// TwinCAT 3 PLC project AnalysisPLC
// ProgramVersion: 3.1.4023.0
// libraries:
//   Tc2_EtherCAT, * (Beckhoff Automation GmbH)
//   Tc2_Standard, * (Beckhoff Automation GmbH)
//   Tc2_System, * (Beckhoff Automation GmbH)
//   Tc2_Utilities, * (Beckhoff Automation GmbH)
//   Tc3_Analytics, * (Beckhoff Automation GmbH)
//   Tc3_EventLogger, * (Beckhoff Automation GmbH)
//   Tc3_Module, * (Beckhoff Automation GmbH)
// project tree:
//   / AnalyticsTask.TcTTO, AnalyticsTask_V1_C1.TcTTO, PlcTask.TcTTO
//   DUTs/Analytics/ E_AnalysisComponents.TcDUT, E_DataSourceState.TcDUT, ST_AnalysisReset.TcDUT
//   DUTs/Analytics/HMI/DataSourcePage/ ST_HMI_DataSourceConfig.TcDUT, ST_HMI_DataSourceCtrl.TcDUT, ST_HMI_DataSourceHist.TcDUT, ST_HMI_DataSourceHistInfo.TcDUT, ST_HMI_DataSourceHistRecordInfo.TcDUT, ST_HMI_DataSourceLive.TcDUT, ST_HMI_DataSourceStream.TcDUT
//   DUTs/Analytics/HMI/ ST_HMI_MapItem.TcDUT, ST_HMI_N1_Network.TcDUT, ST_KeyValuePair.TcDUT
//   GVLs/ Analytics.TcGVL, AnalyticsHMI.TcGVL
//   POUs/Analytics/DataSource/Interfaces/ I_DataSource.TcIO, I_VirtualInputSource.TcIO
//   POUs/Analytics/DataSource/Interfaces/VirtualInputSources/ I_V1_Virtual_Input_Source_1.TcIO
//   POUs/Analytics/DataSource/T01 DataSource/ FB_T1_DataSource.TcPOU
//   POUs/Analytics/ FB_Analysis.TcPOU
//   POUs/Analytics/Networks/N01 Network/ FB_N1_Network.TcPOU
//   POUs/Analytics/Networks/N01 Network/Modules/ FB_N1_M1_LifetimeAnalysis1Ch.TcPOU, FB_N1_M2_ThresholdStringClassifier1Ch.TcPOU, FB_N1_M3_TrendLine.TcPOU
//   POUs/Analytics/[Helper]/ F_AlyTimestampToDCTimestruct.TcPOU, F_AlyTimestampToFileTime.TcPOU, F_DCTimestructToFileTime.TcPOU, F_FileTimeToDCTimestruct.TcPOU
//   POUs/ MAIN.TcPOU, MAIN_Analytics.TcPOU, MAIN_Analytics_V1_C1.TcPOU

CONFIGURATION AnalysisPLC
    RESOURCE PLC ON TwinCAT3
        TASK AnalyticsTask(INTERVAL := T#10ms, PRIORITY := 21);
        TASK AnalyticsTask_V1_C1(INTERVAL := T#10ms, PRIORITY := 1);
        TASK PlcTask(INTERVAL := T#10ms, PRIORITY := 20);
        PROGRAM MAIN_Analytics WITH AnalyticsTask : MAIN_Analytics;
        PROGRAM MAIN_Analytics_V1_C1 WITH AnalyticsTask_V1_C1 : MAIN_Analytics_V1_C1;
        PROGRAM MAIN WITH PlcTask : MAIN;
    END_RESOURCE
END_CONFIGURATION

// ---- DUTs/Analytics/E_AnalysisComponents.TcDUT
{attribute 'qualified_only'}
{attribute 'strict'}
TYPE E_AnalysisComponents : 
(
	All := -1,
	N1_Network := 0,
	N1_M1_LifetimeAnalysis1Ch := 1,
	N1_M2_ThresholdStringClassifier1Ch := 2,
	N1_M3_TrendLine := 3
) ;
END_TYPE

// ---- DUTs/Analytics/E_DataSourceState.TcDUT
{attribute 'qualified_only'}
{attribute 'strict'}
TYPE E_DataSourceState : 
(
	eUnknown := 0,
	eNotConnected,
	eReceiveData,
	eReceiveData_Cancel,
	eReceiveData_Pause,
	eError
) ;
END_TYPE

// ---- DUTs/Analytics/HMI/DataSourcePage/ST_HMI_DataSourceConfig.TcDUT
TYPE ST_HMI_DataSourceConfig : 
STRUCT
	nID: DINT;
	sName: STRING(80);
	sDisplayName: STRING(80);
	nStreamCount: INT;
	aStreams: ARRAY [0..9] OF ST_HMI_DataSourceStream;
END_STRUCT
END_TYPE

// ---- DUTs/Analytics/HMI/DataSourcePage/ST_HMI_DataSourceCtrl.TcDUT
TYPE ST_HMI_DataSourceCtrl : 
STRUCT
	nActiveMachineIdx: INT;
	nActiveStreamIdx: INT;
	
	bHistorical: BOOL;
	
	//IF Historical
	nActiveRecordIdx: INT;
	
	dtSelectedRangeStart: DCTIMESTRUCT;
	dtSelectedRangeEnd: DCTIMESTRUCT;
	
	bStart: BOOL;
	bCancel: BOOL;
	bPause: BOOL;
	
	bUpdateRecordList: BOOL;
END_STRUCT
END_TYPE

// ---- DUTs/Analytics/HMI/DataSourcePage/ST_HMI_DataSourceHist.TcDUT
TYPE ST_HMI_DataSourceHist : 
STRUCT
	dtCurrentTimestamp: DCTIMESTRUCT;
	nCurrentRecordID: DINT;
	sDisplayName: STRING(80);
	stSourceInfo: ST_HMI_DataSourceHistInfo;
	nRecordCount: DINT;
	aRecords: ARRAY [0..255] OF ST_HMI_DataSourceHistRecordInfo;
END_STRUCT
END_TYPE

// ---- DUTs/Analytics/HMI/DataSourcePage/ST_HMI_DataSourceHistInfo.TcDUT
TYPE ST_HMI_DataSourceHistInfo : 
STRUCT
	sSPGuid: GUID;
	sAlyFilePath: STRING(255);
	sSourceType: STRING(80);
	sTopic: STRING(255);
	sLayoutID: GUID;
END_STRUCT
END_TYPE

// ---- DUTs/Analytics/HMI/DataSourcePage/ST_HMI_DataSourceHistRecordInfo.TcDUT
TYPE ST_HMI_DataSourceHistRecordInfo : 
STRUCT
	nID: DINT;
	sName: STRING(80);
	sDisplayName: STRING(80);
	dtRecordStart: DCTIMESTRUCT;
	dtRecordEnd: DCTIMESTRUCT;
	dtSelectedRangeStart: DCTIMESTRUCT;
	dtSelectedRangeEnd: DCTIMESTRUCT;
END_STRUCT
END_TYPE

// ---- DUTs/Analytics/HMI/DataSourcePage/ST_HMI_DataSourceLive.TcDUT
TYPE ST_HMI_DataSourceLive : 
STRUCT
	dtLiveTimestamp: DCTIMESTRUCT;
	sDisplayName: STRING(80);
END_STRUCT
END_TYPE

// ---- DUTs/Analytics/HMI/DataSourcePage/ST_HMI_DataSourceStream.TcDUT
TYPE ST_HMI_DataSourceStream : 
STRUCT
	sSource: STRING(80);
	sStreamSystemID: GUID;
	sTopic: STRING(255);
	stLive: ST_HMI_DataSourceLive;
	stHist: ST_HMI_DataSourceHist;
END_STRUCT
END_TYPE

// ---- DUTs/Analytics/HMI/ST_HMI_MapItem.TcDUT
TYPE ST_HMI_MapItem : 
STRUCT
	sName: T_MaxString;
	sDescription: T_MaxString;
	sPosition: T_MaxString;
	nStatus: INT;
END_STRUCT
END_TYPE

// ---- DUTs/Analytics/HMI/ST_HMI_N1_Network.TcDUT
TYPE ST_HMI_N1_Network : 
STRUCT
	//Lifetime Analysis 1Ch
	tM1_fbLifetimeElapsed: ST_ALY_TimeSpan; //Elapsed (Times)
	tM1_fbLifetimeRemaining: ST_ALY_TimeSpan; //Remaining (Times)
	
	//Threshold String Classifier 1Ch
	sM2_sStringLevel1: STRING(255); //ConfigLevel1
	sM2_sStringLevel2: STRING(255); //ConfigLevel2
	sM2_sStringLevel3: STRING(255); //ConfigLevel3
	sM2_sResult: STRING(255); //String Classification
	fM2_nDataIn: LREAL; //Value
	
	//Trend Line
	aM3_aTrendData: ARRAY [1..1] OF ARRAY [1..10080] OF LREAL; //RawData
	dtM3_fbLastValue: DCTIMESTRUCT; //LastValueTimestamp
	nM3_nCountValues: DINT; //CountedValues
	aM3_aChannelNames: ARRAY [0..0] OF STRING(255); //DisplayNames
END_STRUCT
END_TYPE

// ---- DUTs/Analytics/HMI/ST_KeyValuePair.TcDUT
TYPE ST_KeyValuePair : 
STRUCT
	sKey: STRING(255);
	sValue: STRING(255);
END_STRUCT
END_TYPE

// ---- DUTs/Analytics/ST_AnalysisReset.TcDUT
TYPE ST_AnalysisReset : 
STRUCT
	eResetComponent: E_AnalysisComponents := E_AnalysisComponents.All;
	bResetExecute: BOOL;
END_STRUCT
END_TYPE

// ---- GVLs/Analytics.TcGVL
{attribute 'qualified_only'}
VAR_GLOBAL
	//DataSources
	fbT1_DataSource: FB_T1_DataSource;
	
	bLock_T1: BOOL;
	
	stReset: ST_AnalysisReset;
END_VAR

// ---- GVLs/AnalyticsHMI.TcGVL
{attribute 'qualified_only'}
VAR_GLOBAL
	//Switch between historical and live data
	stHMI_DataSourceCtrl: ST_HMI_DataSourceCtrl;
	stHMI_DataSourceConfig: ARRAY [0..0] OF ST_HMI_DataSourceConfig := [
											(nID:= 1, sName:= 'fbT1_DataSource', sDisplayName:= 'b375d0e8-9412-9d91-04c5-b1a76c1b6bbd', nStreamCount:= 1,
												aStreams:=[(sSource:= 'TwinCAT Analytics Logger', sStreamSystemID:= STRING_TO_GUID('b375d0e8-9412-9d91-04c5-b1a76c1b6bbd'), sTopic:= 'DefaultMainTopic/PlcStream1',
													stLive:= (sDisplayName:= 'DataSource T1')
														)])
											];
	
	//Reset
	
	//HMI Structs
	stHMI_N1_Network: ST_HMI_N1_Network;
	
	//HMI Map Items
	aMapItems: ARRAY [0..0] OF ST_HMI_MapItem := [(sName:='b375d0e8-9412-9d91-04c5-b1a76c1b6bbd', sDescription:='', sPosition:='', nStatus:= 0)];
END_VAR

// ---- POUs/Analytics/DataSource/Interfaces/I_DataSource.TcIO
INTERFACE I_DataSource

METHOD Call : BOOL
END_METHOD

METHOD GetData : BOOL
VAR_INPUT
	nElement: UDINT;
END_VAR
END_METHOD

METHOD HistoricalCtrl : BOOL
VAR_INPUT
	stCtrl: REFERENCE TO ST_HMI_DataSourceCtrl;
	stHistStreamInfo: REFERENCE TO ST_HMI_DataSourceHist;
	stRecordInfo: REFERENCE TO ST_HMI_DataSourceHistRecordInfo;
END_VAR
END_METHOD

METHOD UpdateRecordList : BOOL
VAR_INPUT
	stCtrl: REFERENCE TO ST_HMI_DataSourceCtrl;
	sStreamSystemID: GUID;
	stHistStreamInfo: REFERENCE TO ST_HMI_DataSourceHist;
END_VAR
END_METHOD

METHOD NewDataAvailable : BOOL
VAR_INPUT
	nLastDataHandle: ULINT;
END_VAR
END_METHOD

PROPERTY nDataHandle : ULINT
GET
END_GET
END_PROPERTY

PROPERTY nElements : UDINT
GET
END_GET
END_PROPERTY

PROPERTY dtTimestamp : DCTIMESTRUCT
GET
END_GET
END_PROPERTY

END_INTERFACE

// ---- POUs/Analytics/DataSource/Interfaces/I_VirtualInputSource.TcIO
INTERFACE I_VirtualInputSource

PROPERTY tTimestamp : ULINT
GET
END_GET
END_PROPERTY

PROPERTY bNewData : BOOL
GET
END_GET
END_PROPERTY

END_INTERFACE

// ---- POUs/Analytics/DataSource/Interfaces/VirtualInputSources/I_V1_Virtual_Input_Source_1.TcIO
INTERFACE I_V1_Virtual_Input_Source_1 EXTENDS I_VirtualInputSource

PROPERTY bV1_Virtual_Input : BOOL
GET
END_GET
END_PROPERTY

PROPERTY nV1_Virtual_Input_1 : INT
GET
END_GET
END_PROPERTY

END_INTERFACE

// ---- POUs/MAIN_Analytics.TcPOU
PROGRAM MAIN_Analytics
VAR
	sCurrentStreamSystemID: GUID;
	stHistStreamInfo: REFERENCE TO ST_HMI_DataSourceHist;
	stHistRecordInfo: REFERENCE TO ST_HMI_DataSourceHistRecordInfo;
END_VAR



//Call DataSource FBs
IF MAIN_Analytics_V1_C1.nLastDataHandle = Analytics.fbT1_DataSource.nDataHandle THEN
	Analytics.fbT1_DataSource.Call();
END_IF



//Map to HMI
CASE AnalyticsHMI.stHMI_DataSourceCtrl.nActiveMachineIdx OF
	0:
		MAIN_Analytics_V1_C1.A_MapToHMI();
END_CASE

END_PROGRAM

// ---- POUs/MAIN_Analytics_V1_C1.TcPOU
PROGRAM MAIN_Analytics_V1_C1
VAR_OUTPUT
	bError: BOOL;
	ipTcResult: I_TcMessage;
	nLastDataHandle: ULINT;
END_VAR
VAR
	fbAnalysis: FB_Analysis;
	
	nElement: UDINT;
	nSample: UDINT;
END_VAR

IF TestAndSet(Analytics.bLock_T1) THEN
	IF Analytics.fbT1_DataSource.NewDataAvailable(nLastDataHandle) THEN
		FOR nElement:= 1 TO Analytics.fbT1_DataSource.nElements BY 1 DO
			IF Analytics.fbT1_DataSource.GetData(nElement) THEN

				fbAnalysis.Call(Analytics.fbT1_DataSource);
				IF fbAnalysis.bError THEN
					EXIT;
				END_IF
			END_IF
		END_FOR
		nLastDataHandle:= Analytics.fbT1_DataSource.nDataHandle;
	ELSE
		fbAnalysis.Call(0);
	END_IF
	Analytics.bLock_T1:= FALSE;
END_IF

//Error Handling
bError:= fbAnalysis.bError;
ipTcResult:= fbAnalysis.ipTcResult;

ACTION A_MapToHMI:

//Map HMI Current Timestamp
AnalyticsHMI.stHMI_DataSourceConfig[0].aStreams[0].stLive.dtLiveTimestamp:= Analytics.fbT1_DataSource.dtTimestamp;

//Map In-/Outputs of the Analysis to HMI Structs
fbAnalysis.fbN1_Network.SetHMIValues(ADR(AnalyticsHMI.stHMI_N1_Network));
END_ACTION

END_PROGRAM

// ---- POUs/Analytics/FB_Analysis.TcPOU
FUNCTION_BLOCK FB_Analysis
VAR_INPUT
	fbN1_Network: FB_N1_Network;
END_VAR
VAR_OUTPUT
	bError: BOOL;
	ipTcResult: I_TcMessage;
END_VAR
VAR
	R_TRIG_Reset: R_TRIG;
	bResetBusy: BOOL;
	
	_tTimestamp: ULINT;
END_VAR

METHOD Call : BOOL
VAR_INPUT
	ipVirtual_Input_Source_1: I_V1_Virtual_Input_Source_1;
END_VAR
VAR
END_VAR

IF ipVirtual_Input_Source_1 <> 0 THEN

	_tTimestamp:= ipVirtual_Input_Source_1.tTimestamp;

	//Analytics Network "Network" with ID: 1
	fbN1_Network.Call(ipVirtual_Input_Source_1);


	//Error Handling
	IF fbN1_Network.bError THEN
		bError:= TRUE;
		ipTcResult:= fbN1_Network.ipTcResult;
	ELSE
		bError:= FALSE;
	END_IF
END_IF
END_METHOD

PROPERTY tTimestamp : ULINT
GET
tTimestamp:= _tTimestamp;
END_GET
END_PROPERTY

END_FUNCTION_BLOCK

// ---- POUs/Analytics/Networks/N01 Network/FB_N1_Network.TcPOU
//Analytics Network "Network" with ID: 1
{attribute 'no_assign'}
FUNCTION_BLOCK FB_N1_Network
VAR_INPUT
	fbM1_LifetimeAnalysis1Ch: FB_N1_M1_LifetimeAnalysis1Ch;
	fbM2_ThresholdStringClassifier1Ch: FB_N1_M2_ThresholdStringClassifier1Ch;
	fbM3_TrendLine: FB_N1_M3_TrendLine;
END_VAR
VAR_OUTPUT
	bError: BOOL;
	ipTcResult: I_TcMessage;
END_VAR
VAR
END_VAR

METHOD Call : BOOL
VAR_INPUT
	ipVirtual_Input_Source_1: I_V1_Virtual_Input_Source_1;
END_VAR
VAR
END_VAR

ValueMapping(ipVirtual_Input_Source_1);

//The Lifetime Analysis 1Ch calculates the elapsed and the estimated remaining lifetime of a device. The input channel should provide boolean values so that every switching procedure represents a cycle which can be converted into the elapsed lifetime. Optional a boolean signal for Enable Execution can be selected, so that the algorithm is just active if the value of the selected signal is TRUE.
fbM1_LifetimeAnalysis1Ch.Call(SEL(ipVirtual_Input_Source_1 <> 0, FALSE, ipVirtual_Input_Source_1.bNewData));

//The Threshold String Classifier 1Ch classifies the input values into three different classes according to the configured thresholds. The class names (output strings) can be configured individually as String 1, String 2 and String 3. Optional a boolean signal for Enable Execution can be selected, so that the algorithm is just active if the value of the selected signal is TRUE.
fbM2_ThresholdStringClassifier1Ch.Call(SEL(ipVirtual_Input_Source_1 <> 0, FALSE, ipVirtual_Input_Source_1.bNewData));

//This Module is used for the One-click Dashboard to generate a special analytics trend chart.
fbM3_TrendLine.Call(SEL(ipVirtual_Input_Source_1 <> 0, FALSE, ipVirtual_Input_Source_1.bNewData));

//Error Handling
IF fbM1_LifetimeAnalysis1Ch.bError THEN
	bError:= TRUE;
	ipTcResult:= fbM1_LifetimeAnalysis1Ch.ipTcResult;
ELSIF fbM2_ThresholdStringClassifier1Ch.bError THEN
	bError:= TRUE;
	ipTcResult:= fbM2_ThresholdStringClassifier1Ch.ipTcResult;
ELSIF fbM3_TrendLine.bError THEN
	bError:= TRUE;
	ipTcResult:= fbM3_TrendLine.ipTcResult;
ELSE
	bError:= FALSE;
END_IF
END_METHOD

METHOD Reset : BOOL
VAR
	bResult: BOOL := TRUE;
END_VAR

bResult:= bResult AND fbM1_LifetimeAnalysis1Ch.Reset();
bResult:= bResult AND fbM2_ThresholdStringClassifier1Ch.Reset();
bResult:= bResult AND fbM3_TrendLine.Reset();
Reset:= bResult;
END_METHOD

METHOD SetHMIValues : BOOL
VAR_INPUT
	pHMI_N1_Network: POINTER TO ST_HMI_N1_Network;
END_VAR
VAR
END_VAR

//Modules
fbM1_LifetimeAnalysis1Ch.SetHMI(pHMI_N1_Network);
fbM2_ThresholdStringClassifier1Ch.SetHMI(pHMI_N1_Network);
fbM3_TrendLine.SetHMI(pHMI_N1_Network);

SetHMIValues:= TRUE;
END_METHOD

METHOD PRIVATE ValueMapping : BOOL
VAR_INPUT
	ipVirtual_Input_Source_1: I_V1_Virtual_Input_Source_1;
END_VAR
VAR
END_VAR
//Module fbM1_LifetimeAnalysis1Ch
fbM1_LifetimeAnalysis1Ch.tTimestamp:= ipVirtual_Input_Source_1.tTimestamp;
fbM1_LifetimeAnalysis1Ch.bDataIn:= ipVirtual_Input_Source_1.bV1_Virtual_Input;

//Module fbM2_ThresholdStringClassifier1Ch
fbM2_ThresholdStringClassifier1Ch.tTimestamp:= ipVirtual_Input_Source_1.tTimestamp;
fbM2_ThresholdStringClassifier1Ch.nDataIn:= ipVirtual_Input_Source_1.nV1_Virtual_Input_1;

//Module fbM3_TrendLine
fbM3_TrendLine.tTimestamp:= ipVirtual_Input_Source_1.tTimestamp;
fbM3_TrendLine.nDataInCh1:= ipVirtual_Input_Source_1.nV1_Virtual_Input_1;
END_METHOD

END_FUNCTION_BLOCK

// ---- POUs/Analytics/Networks/N01 Network/Modules/FB_N1_M1_LifetimeAnalysis1Ch.TcPOU
//The Lifetime Analysis 1Ch calculates the elapsed and the estimated remaining lifetime of a device. The input channel should provide boolean values so that every switching procedure represents a cycle which can be converted into the elapsed lifetime. Optional a boolean signal for Enable Execution can be selected, so that the algorithm is just active if the value of the selected signal is TRUE.
FUNCTION_BLOCK FB_N1_M1_LifetimeAnalysis1Ch
VAR_INPUT
	bDataIn: BOOL;
	tTimestamp: ULINT;
	bEnableExecution: BOOL := TRUE;
	bReset: BOOL;
	bReconfigure: BOOL := TRUE;
	stThresholdLevel: ST_ALY_Threshold;
	tLifetimeEstimated: LTIME;
END_VAR
VAR_OUTPUT
	bError: BOOL;
	ipTcResult: I_TcMessage;
	bNewResult: BOOL;
	fbLifetimeElapsed: FB_ALY_TimeSpan;
	fbLifetimeRemaining: FB_ALY_TimeSpan;
END_VAR
VAR
	
	bConfigured: BOOL;
	R_TRIG_Reconfigure: R_TRIG;
	
	fbALY_LifeTimeAnalysis_1Ch: FB_ALY_LifeTimeAnalysis_1Ch;
END_VAR

METHOD Call : BOOL
VAR_INPUT
	bNewData: BOOL;
END_VAR
VAR
END_VAR
IF NOT bConfigured THEN
	bConfigured:= TRUE;

	tLifetimeEstimated:= LTIME#1h;

	//stThresholdLevel
	stThresholdLevel.eComparisonOperator:= E_ALY_ComparisonOperator.NotEqualTo;
	stThresholdLevel.fThreshold:= 0;

END_IF

R_TRIG_Reconfigure(CLK:= bReconfigure);
IF R_TRIG_Reconfigure.Q THEN
	fbALY_LifeTimeAnalysis_1Ch.ConfigureChannel(stThresholdLevel:=stThresholdLevel);

	fbALY_LifeTimeAnalysis_1Ch.Configure(tLifetimeEstimated:=tLifetimeEstimated);

	bReconfigure:= FALSE;
END_IF

IF bReset THEN
	Reset();
END_IF

IF bEnableExecution THEN
	IF bNewData THEN
		fbALY_LifeTimeAnalysis_1Ch.SetChannelValue(Input:=bDataIn);

		fbALY_LifeTimeAnalysis_1Ch.Call(tTimestamp:=tTimestamp);

		bNewResult:= fbALY_LifeTimeAnalysis_1Ch.bNewResult;
		fbLifetimeElapsed:= fbALY_LifeTimeAnalysis_1Ch.fbLifetimeElapsed;
		fbLifetimeRemaining:= fbALY_LifeTimeAnalysis_1Ch.fbLifetimeRemaining;

		bError:= fbALY_LifeTimeAnalysis_1Ch.bError;
		ipTcResult:= fbALY_LifeTimeAnalysis_1Ch.ipResultMessage;
	END_IF
END_IF
END_METHOD

METHOD Reset : BOOL
VAR
END_VAR
Reset:= fbALY_LifeTimeAnalysis_1Ch.Reset();

bNewResult:= fbALY_LifeTimeAnalysis_1Ch.bNewResult;
fbLifetimeElapsed:= fbALY_LifeTimeAnalysis_1Ch.fbLifetimeElapsed;
fbLifetimeRemaining:= fbALY_LifeTimeAnalysis_1Ch.fbLifetimeRemaining;

bError:= NOT Reset;
ipTcResult:= fbALY_LifeTimeAnalysis_1Ch.ipResultMessage;
END_METHOD

METHOD SetHMI : BOOL
VAR_INPUT
	pHMI_N1_Network: POINTER TO ST_HMI_N1_Network;
END_VAR
VAR
END_VAR

pHMI_N1_Network^.tM1_fbLifetimeElapsed:= fbLifetimeElapsed.stStructured;
pHMI_N1_Network^.tM1_fbLifetimeRemaining:= fbLifetimeRemaining.stStructured;
END_METHOD

END_FUNCTION_BLOCK

// ---- POUs/Analytics/Networks/N01 Network/Modules/FB_N1_M2_ThresholdStringClassifier1Ch.TcPOU
//The Threshold String Classifier 1Ch classifies the input values into three different classes according to the configured thresholds. The class names (output strings) can be configured individually as String 1, String 2 and String 3. Optional a boolean signal for Enable Execution can be selected, so that the algorithm is just active if the value of the selected signal is TRUE.
FUNCTION_BLOCK FB_N1_M2_ThresholdStringClassifier1Ch
VAR_INPUT
	nDataIn: INT;
	tTimestamp: ULINT;
	bEnableExecution: BOOL := TRUE;
	bReset: BOOL;
	bReconfigure: BOOL := TRUE;
	fThresholdLevel12: LREAL;
	fThresholdLevel23: LREAL;
	sStringLevel1: STRING(255);
	sStringLevel2: STRING(255);
	sStringLevel3: STRING(255);
END_VAR
VAR_OUTPUT
	bError: BOOL;
	ipTcResult: I_TcMessage;
	bNewResult: BOOL;
	sResult: STRING(255);
	fbTimeLastEvent: FB_ALY_DateTime;
END_VAR
VAR
	
	bConfigured: BOOL;
	R_TRIG_Reconfigure: R_TRIG;
	
	fbALY_ThresholdStringClassificator_1Ch: FB_ALY_ThresholdStringClassificator_1Ch;
END_VAR

METHOD Call : BOOL
VAR_INPUT
	bNewData: BOOL;
END_VAR
VAR
END_VAR
IF NOT bConfigured THEN
	bConfigured:= TRUE;

	fThresholdLevel12:= 20000;
	fThresholdLevel23:= 28000;
	sStringLevel1:= 'Normal';
	sStringLevel2:= 'High';
	sStringLevel3:= 'High High';

END_IF

R_TRIG_Reconfigure(CLK:= bReconfigure);
IF R_TRIG_Reconfigure.Q THEN
	fbALY_ThresholdStringClassificator_1Ch.Configure(
		fThresholdLevel12:= fThresholdLevel12,
		fThresholdLevel23:= fThresholdLevel23,
		sStringLevel1:= sStringLevel1,
		sStringLevel2:= sStringLevel2,
		sStringLevel3:= sStringLevel3);

	bReconfigure:= FALSE;
END_IF

IF bReset THEN
	Reset();
END_IF

IF bEnableExecution THEN
	IF bNewData THEN
		fbALY_ThresholdStringClassificator_1Ch.SetChannelValue(Input:=nDataIn);

		fbALY_ThresholdStringClassificator_1Ch.Call(tTimestamp:=tTimestamp);

		bNewResult:= fbALY_ThresholdStringClassificator_1Ch.bNewResult;
		sResult:= fbALY_ThresholdStringClassificator_1Ch.sResult;
		fbTimeLastEvent:= fbALY_ThresholdStringClassificator_1Ch.fbTimeLastEvent;

		bError:= fbALY_ThresholdStringClassificator_1Ch.bError;
		ipTcResult:= fbALY_ThresholdStringClassificator_1Ch.ipResultMessage;
	END_IF
END_IF
END_METHOD

METHOD Reset : BOOL
VAR
END_VAR
Reset:= fbALY_ThresholdStringClassificator_1Ch.Reset();

bNewResult:= fbALY_ThresholdStringClassificator_1Ch.bNewResult;
sResult:= fbALY_ThresholdStringClassificator_1Ch.sResult;
fbTimeLastEvent:= fbALY_ThresholdStringClassificator_1Ch.fbTimeLastEvent;

bError:= NOT Reset;
ipTcResult:= fbALY_ThresholdStringClassificator_1Ch.ipResultMessage;
END_METHOD

METHOD SetHMI : BOOL
VAR_INPUT
	pHMI_N1_Network: POINTER TO ST_HMI_N1_Network;
END_VAR
VAR
END_VAR

pHMI_N1_Network^.sM2_sStringLevel1:= sStringLevel1;
pHMI_N1_Network^.sM2_sStringLevel2:= sStringLevel2;
pHMI_N1_Network^.sM2_sStringLevel3:= sStringLevel3;
pHMI_N1_Network^.sM2_sResult:= sResult;
pHMI_N1_Network^.fM2_nDataIn:= TO_LREAL(nDataIn);
END_METHOD

END_FUNCTION_BLOCK

// ---- POUs/Analytics/Networks/N01 Network/Modules/FB_N1_M3_TrendLine.TcPOU
//This Module is used for the One-click Dashboard to generate a special analytics trend chart.
FUNCTION_BLOCK FB_N1_M3_TrendLine
VAR_INPUT
	nDataInCh1: INT;
	tTimestamp: ULINT;
	bEnableExecution: BOOL := TRUE;
	bReset: BOOL;
	bReconfigure: BOOL := TRUE;
	aChannelNames: ARRAY [0..0] OF STRING(255);
END_VAR
VAR_OUTPUT
	bError: BOOL;
	ipTcResult: I_TcMessage;
	bNewResult: BOOL;
	aTrendData: ARRAY [1..1] OF ARRAY [1..10080] OF LREAL;
	fbLastValue: FB_ALY_DateTime;
	nCountValues: UDINT;
END_VAR
VAR
	nNumChannels: INT := 1;
	
	bConfigured: BOOL;
	R_TRIG_Reconfigure: R_TRIG;
	
	fbALY_TrendLine: FB_ALY_TrendLine(nNumChannels:=nNumChannels);
END_VAR

METHOD Call : BOOL
VAR_INPUT
	bNewData: BOOL;
END_VAR
VAR
END_VAR
IF NOT bConfigured THEN
	bConfigured:= TRUE;

	aChannelNames[0]:= 'Resistor';

END_IF

R_TRIG_Reconfigure(CLK:= bReconfigure);
IF R_TRIG_Reconfigure.Q THEN

	bReconfigure:= FALSE;
END_IF

IF bReset THEN
	Reset();
END_IF

IF bEnableExecution THEN
	IF bNewData THEN
		fbALY_TrendLine.SetChannelValue(nChannel:=1, Input:=nDataInCh1);

		fbALY_TrendLine.Call(tTimestamp:=tTimestamp);

		bNewResult:= fbALY_TrendLine.bNewResult;
		fbLastValue:= fbALY_TrendLine.fbLastValue;
		nCountValues:= fbALY_TrendLine.nCountValues;

		fbALY_TrendLine.GetChannelOutputArray(nChannel:=1, pArrayOut:=ADR(aTrendData[1]), nArrayOutSize:=SIZEOF(aTrendData[1]));

		bError:= fbALY_TrendLine.bError;
		ipTcResult:= fbALY_TrendLine.ipResultMessage;
	END_IF
END_IF
END_METHOD

METHOD Reset : BOOL
VAR
END_VAR
Reset:= fbALY_TrendLine.Reset();

bNewResult:= fbALY_TrendLine.bNewResult;
fbLastValue:= fbALY_TrendLine.fbLastValue;
nCountValues:= fbALY_TrendLine.nCountValues;

fbALY_TrendLine.GetChannelOutputArray(nChannel:=1, pArrayOut:=ADR(aTrendData[1]), nArrayOutSize:=SIZEOF(aTrendData[1]));

bError:= NOT Reset;
ipTcResult:= fbALY_TrendLine.ipResultMessage;
END_METHOD

METHOD SetHMI : BOOL
VAR_INPUT
	pHMI_N1_Network: POINTER TO ST_HMI_N1_Network;
END_VAR
VAR
	i: INT;
END_VAR

FOR i:=1 TO 1 DO
	pHMI_N1_Network^.aM3_aTrendData[i]:= aTrendData[i];
END_FOR
fbLastValue.nUtcTimeBias:= -420; //UTC Offset [(UTC+07:00) Bangkok, Hanoi, Jakarta]
pHMI_N1_Network^.dtM3_fbLastValue:= fbLastValue.stStructured;
pHMI_N1_Network^.nM3_nCountValues:= TO_DINT(nCountValues);
FOR i:=0 TO 0 DO
	pHMI_N1_Network^.aM3_aChannelNames[i]:= aChannelNames[i];
END_FOR
END_METHOD

END_FUNCTION_BLOCK

// ---- POUs/MAIN.TcPOU
PROGRAM MAIN
VAR
END_VAR

END_PROGRAM

// ---- POUs/Analytics/DataSource/T01 DataSource/FB_T1_DataSource.TcPOU
FUNCTION_BLOCK FB_T1_DataSource IMPLEMENTS I_DataSource, I_V1_Virtual_Input_Source_1
VAR_OUTPUT
	eDataState: E_DataSourceState;
END_VAR
VAR
	_bV1_Virtual_Input: BOOL;
	_nV1_Virtual_Input_1: INT;
	_tTimestamp: ULINT;
	
	_nElements: UDINT;
	_nCurrentElement: UDINT;
	
	_nDataHandle: ULINT;
	
	fbIotSymbol_MAIN_bDinx: FB_ALY_IotSymbol_BOOL := (stConfig:= (sSymbolName:= 'MAIN.bDinx'));
	fbIotSymbol_MAIN_nAinx: FB_ALY_IotSymbol_INT := (stConfig:= (sSymbolName:= 'MAIN.nAinx'));
	
	//Target T1 = Broker:"192.168.1.10" Topic:"DefaultMainTopic/PlcStream1"
	fbStreamHelper: FB_ALY_StreamHelper;
	bConfigured: BOOL := FALSE;
	
	fbALY_GetSystemTime: FB_ALY_GetSystemTime;
END_VAR

PROPERTY bNewData : BOOL
GET
bNewData:= _nElements > 0;
END_GET
END_PROPERTY

PROPERTY bV1_Virtual_Input : BOOL
GET
bV1_Virtual_Input:= _bV1_Virtual_Input;
END_GET
END_PROPERTY

METHOD Call : BOOL
VAR
	stConfig: ST_ALY_StreamHelper_Config;
END_VAR
IF NOT fbStreamHelper.bConfigured THEN
	stConfig.nObjectID:= 16#01010010;
	stConfig.nNumInputBuffer:= 20;
	fbStreamHelper.Configure(stConfig);
END_IF

IF NOT bConfigured THEN
	//MAIN.bDinx
	fbStreamHelper.AddIotSymbol(fbIotSymbol_MAIN_bDinx);
	//MAIN.nAinx
	fbStreamHelper.AddIotSymbol(fbIotSymbol_MAIN_nAinx);

	bConfigured:= TRUE;
END_IF

fbStreamHelper.Call();
IF fbStreamHelper.bError THEN
	eDataState:= E_DataSourceState.eError;
ELSIF NOT fbStreamHelper.bConnected THEN
	eDataState:= E_DataSourceState.eNotConnected;
ELSE
	IF eDataState <> E_DataSourceState.eReceiveData_Cancel AND eDataState <> E_DataSourceState.eReceiveData_Pause THEN
		eDataState:= E_DataSourceState.eReceiveData;
		_nElements:= fbStreamHelper.nNumElements;
	ELSE
		_nElements:= 0;
	END_IF
END_IF

fbALY_GetSystemTime.Call();


IF _nElements > 0 THEN
	_nDataHandle:= _nDataHandle + 1;
END_IF

_nCurrentElement:= 0;
END_METHOD

PROPERTY dtTimestamp : DCTIMESTRUCT
GET

dtTimestamp:= F_AlyTimestampToDCTimestruct(_tTimestamp);
END_GET
END_PROPERTY

METHOD GetData : BOOL
VAR_INPUT
	nElement: UDINT;
END_VAR
VAR
END_VAR
IF nElements > 0 THEN
	IF nElement <= nElements THEN

		IF _nCurrentElement <> nElement THEN
			//Set local raw inputs
			_bV1_Virtual_Input:= fbIotSymbol_MAIN_bDinx.GetValue(nElement);
			_nV1_Virtual_Input_1:= fbIotSymbol_MAIN_nAinx.GetValue(nElement);

			//Set tTimestamp
			_tTimestamp:= fbStreamHelper.GetTimestampElement(nElement);


			_nCurrentElement:= nElement;
		END_IF
	END_IF
	GetData:= TRUE;
ELSE
	GetData:= FALSE;
END_IF
END_METHOD

METHOD HistoricalCtrl : BOOL
VAR_INPUT
	stCtrl: REFERENCE TO ST_HMI_DataSourceCtrl;
	stHistStreamInfo: REFERENCE TO ST_HMI_DataSourceHist;
	stRecordInfo: REFERENCE TO ST_HMI_DataSourceHistRecordInfo;
END_VAR
VAR
END_VAR
//Not implemented
END_METHOD

PROPERTY nDataHandle : ULINT
GET
nDataHandle:= _nDataHandle;
END_GET
END_PROPERTY

PROPERTY nElements : UDINT
GET
nElements:= _nElements;
END_GET
END_PROPERTY

METHOD NewDataAvailable : BOOL
VAR_INPUT
	nLastDataHandle: ULINT;
END_VAR
VAR
END_VAR
NewDataAvailable:= _nElements > 0 AND _nDataHandle <> nLastDataHandle;
END_METHOD

PROPERTY nV1_Virtual_Input_1 : INT
GET
nV1_Virtual_Input_1:= _nV1_Virtual_Input_1;
END_GET
END_PROPERTY

PROPERTY tTimestamp : ULINT
GET
tTimestamp:= _tTimestamp;
END_GET
END_PROPERTY

METHOD UpdateRecordList : BOOL
VAR_INPUT
	stCtrl: REFERENCE TO ST_HMI_DataSourceCtrl;
	sStreamSystemID: GUID;
	stHistStreamInfo: REFERENCE TO ST_HMI_DataSourceHist;
END_VAR
VAR
END_VAR
//Not implemented
END_METHOD

END_FUNCTION_BLOCK

// ---- POUs/Analytics/[Helper]/F_AlyTimestampToDCTimestruct.TcPOU
FUNCTION F_AlyTimestampToDCTimestruct : DCTIMESTRUCT
VAR_INPUT
	tTimestamp: ULINT;
END_VAR
VAR
	tFileTime: T_FILETIME;
	newDCTime: T_DCTIME64;
	
	fbToLocal: FB_FileTimeToTzSpecificLocalTime;
	//(UTC+07:00) Bangkok, Hanoi, Jakarta
	tzInfo: ST_TimeZoneInformation;
END_VAR

tFileTime:= DCTIME64_TO_Filetime(tTimestamp);
fbToLocal(in:= tFileTime, tzInfo:= tzInfo);
newDCTime:= FILETIME_TO_DCTIME64(fbToLocal.out);

F_AlyTimestampToDCTimestruct:= DCTIME64_TO_DCTIMESTRUCT(newDCTime);

END_FUNCTION

// ---- POUs/Analytics/[Helper]/F_AlyTimestampToFileTime.TcPOU
FUNCTION F_AlyTimestampToFileTime : ULINT
VAR_INPUT
	tTimestamp: ULINT;
END_VAR
VAR
	tFileTime: T_FILETIME;
	
	fbToUTC: FB_TzSpecificLocalTimeToFileTime;
	//(UTC+07:00) Bangkok, Hanoi, Jakarta
	tzInfo: ST_TimeZoneInformation;
END_VAR

tFileTime:= DCTIME64_TO_Filetime(tTimestamp);

fbToUTC(in:= tFileTime, tzInfo:= tzInfo);
F_AlyTimestampToFileTime:= ULARGE_TO_ULINT(ULARGE_INTEGER(fbToUTC.out.dwHighDateTime, fbToUTC.out.dwLowDateTime));

END_FUNCTION

// ---- POUs/Analytics/[Helper]/F_DCTimestructToFileTime.TcPOU
FUNCTION F_DCTimestructToFileTime : ULINT
VAR_INPUT
	dtTimestamp: DCTIMESTRUCT;
END_VAR
VAR
	dcTime: T_DCTIME64;
END_VAR

dcTime:= DCTIMESTRUCT_TO_DCTIME64(dtTimestamp);
F_DCTimestructToFileTime:= F_AlyTimestampToFileTime(dcTime);

END_FUNCTION

// ---- POUs/Analytics/[Helper]/F_FileTimeToDCTimestruct.TcPOU
FUNCTION F_FileTimeToDCTimestruct : DCTIMESTRUCT
VAR_INPUT
	tTimestamp: ULINT;
END_VAR
VAR
	tULarge: T_ULARGE_INTEGER;
	tFileTime: T_FILETIME;
	newDCTime: T_DCTIME64;
	
	fbToLocal: FB_FileTimeToTzSpecificLocalTime;
	//(UTC+07:00) Bangkok, Hanoi, Jakarta
	tzInfo: ST_TimeZoneInformation;
END_VAR

tULarge:= ULINT_TO_ULARGE(tTimestamp);
tFileTime.dwLowDateTime:= tULarge.dwLowPart;
tFileTime.dwHighDateTime:= tULarge.dwHighPart;

fbToLocal(in:= tFileTime, tzInfo:= tzInfo);
newDCTime:= FILETIME_TO_DCTIME64(fbToLocal.out);

F_FileTimeToDCTimestruct:= DCTIME64_TO_DCTIMESTRUCT(newDCTime);

END_FUNCTION
